(* This is a comment 1
	with multiple lines
*)
FUNCTION_BLOCK SystemParametersFB
VAR_IN_OUT
	Parameters: GreenMasterBaseParameters;
END_VAR
VAR_INPUT
	Operation: SystemOperationParameters;
	Defrost: DefrostParameters;
	Exercise: ExerciseParameters;
	SystemTime: string;
	{attribute 'TcEncoding':='UTF-8'}
	Diagram: string[8000];
END_VAR
VAR_OUTPUT
END_VAR
VAR
END_VAR

Exercise(Parameters := Parameters);
Operation.ENO := Operation.State > SystemStates.Idle;
Operation.TimeChannels.TC01();
Operation.TimeChannels.TC02();
Operation.TimeChannels.TC03();
Operation.TimeChannels.TC04();
Operation.TimeChannels.TC05();
Operation.TimeChannels.TC06();
Operation.TimeChannels.TC07();

Operation.TimeChannels.TC11();
Operation.TimeChannels.TC12();
Operation.TimeChannels.TC13();
Operation.TimeChannels.TC14();
Operation.TimeChannels.TC15();
Operation.TimeChannels.TC16();
Operation.TimeChannels.TC17();

Operation.TimeChannels.TC21();
Operation.TimeChannels.TC22();
Operation.TimeChannels.TC23();
Operation.TimeChannels.TC24();
Operation.TimeChannels.TC25();
Operation.TimeChannels.TC26();
Operation.TimeChannels.TC27();

Operation.TimeChannels.Q :=
	Operation.TimeChannels.TC01.Q OR
	Operation.TimeChannels.TC02.Q OR
	Operation.TimeChannels.TC03.Q OR
	Operation.TimeChannels.TC04.Q OR
	Operation.TimeChannels.TC05.Q OR
	Operation.TimeChannels.TC06.Q OR
	Operation.TimeChannels.TC07.Q OR
	Operation.TimeChannels.TC11.Q OR
	Operation.TimeChannels.TC12.Q OR
	Operation.TimeChannels.TC13.Q OR
	Operation.TimeChannels.TC14.Q OR
	Operation.TimeChannels.TC15.Q OR
	Operation.TimeChannels.TC16.Q OR
	Operation.TimeChannels.TC17.Q OR
	Operation.TimeChannels.TC21.Q OR
	Operation.TimeChannels.TC22.Q OR
	Operation.TimeChannels.TC23.Q OR
	Operation.TimeChannels.TC24.Q OR
	Operation.TimeChannels.TC25.Q OR
	Operation.TimeChannels.TC26.Q OR
	Operation.TimeChannels.TC27.Q;

Operation.TimeChannelsLocal.TC01();
Operation.TimeChannelsLocal.TC02();
Operation.TimeChannelsLocal.TC03();
Operation.TimeChannelsLocal.TC04();
Operation.TimeChannelsLocal.TC05();
Operation.TimeChannelsLocal.TC06();
Operation.TimeChannelsLocal.TC07();

Operation.TimeChannelsLocal.TC11();
Operation.TimeChannelsLocal.TC12();
Operation.TimeChannelsLocal.TC13();
Operation.TimeChannelsLocal.TC14();
Operation.TimeChannelsLocal.TC15();
Operation.TimeChannelsLocal.TC16();
Operation.TimeChannelsLocal.TC17();

Operation.TimeChannelsLocal.TC21();
Operation.TimeChannelsLocal.TC22();
Operation.TimeChannelsLocal.TC23();
Operation.TimeChannelsLocal.TC24();
Operation.TimeChannelsLocal.TC25();
Operation.TimeChannelsLocal.TC26();
Operation.TimeChannelsLocal.TC27();

Operation.TimeChannelsLocal.Q :=
	Operation.TimeChannelsLocal.TC01.Q OR
	Operation.TimeChannelsLocal.TC02.Q OR
	Operation.TimeChannelsLocal.TC03.Q OR
	Operation.TimeChannelsLocal.TC04.Q OR
	Operation.TimeChannelsLocal.TC05.Q OR
	Operation.TimeChannelsLocal.TC06.Q OR
	Operation.TimeChannelsLocal.TC07.Q OR
	Operation.TimeChannelsLocal.TC11.Q OR
	Operation.TimeChannelsLocal.TC12.Q OR
	Operation.TimeChannelsLocal.TC13.Q OR
	Operation.TimeChannelsLocal.TC14.Q OR
	Operation.TimeChannelsLocal.TC15.Q OR
	Operation.TimeChannelsLocal.TC16.Q OR
	Operation.TimeChannelsLocal.TC17.Q OR
	Operation.TimeChannelsLocal.TC21.Q OR
	Operation.TimeChannelsLocal.TC22.Q OR
	Operation.TimeChannelsLocal.TC23.Q OR
	Operation.TimeChannelsLocal.TC24.Q OR
	Operation.TimeChannelsLocal.TC25.Q OR
	Operation.TimeChannelsLocal.TC26.Q OR
	Operation.TimeChannelsLocal.TC27.Q;

END_FUNCTION_BLOCK

(* stored: Version 1.1.0.1, ProductVersion 3.1.4024.6
   POU SystemParametersFB: Id {f1690a32-b7d9-4c46-bdf1-78c808f8c5e8}, SpecialFunc None *)
